Staubli VAL3: calculateForce.pgx

public program calculateForce(num& x_nDetectValue[], num& x_nFTValue[])
  local num l_nNum
begin

  //This program is used for calculating the interaction force/torque between the robot endeffector and environment
  //based on the detected data and the sensitivity from the sensor.

  //F/T Value=(detected value-zero point value)/main axis sensitivity
  for l_nNum=0 to 5
    x_nFTValue[l_nNum]=(x_nDetectValue[l_nNum]-nZeroPoint[l_nNum])/nSensitivity[l_nNum]
  endFor

end
